(* IEC 61131-3 sources: 89152_FlorisHendrix_AfstudeerProject/89152_FlorisHendrix_ExamenProject/Stations/MachineControl/MachineControl/Class/KTS_Read, 1 file *)

(* ---- KTS_Read.st ---- *)
(*!
<Class
	Name               = "KTS_Read"
	Revision           = "0.0"
	RealtimeTask       = "true"
	DefRealtime        = "10 ms"
	CyclicTask         = "true"
	DefCyclictime      = "50 ms"
	BackgroundTask     = "false"
	Sigmatek           = "false"
	OSInterface        = "false"
	HighPriority       = "false"
	Automatic          = "false"
	UpdateMode         = "Prescan"
	SharedCommandTable = "true"
	Objectsize         = "(624,120)">
	<Channels>
		<Server Name="ClassSvr" Visualized="false" Initialize="false" WriteProtected="true" Retentive="false"/>
		<Server Name="sReadJob" Visualized="true" Initialize="false" WriteProtected="false" Retentive="false"/>
		<Server Name="sRetcode" Visualized="false" Initialize="false" WriteProtected="true" Retentive="false"/>
		<Server Name="sTeach2Points" Visualized="true" Initialize="false" WriteProtected="false" Retentive="false"/>
		<Server Name="sTeachCommand" Visualized="true" Initialize="false" WriteProtected="false" Retentive="false"/>
		<Server Name="sTeachDynamic" Visualized="true" Initialize="false" WriteProtected="false" Retentive="false"/>
		<Server Name="sTeachStart" Visualized="true" Initialize="false" WriteProtected="false" Retentive="false"/>
		<Client Name="coCSVFile" Required="true" Internal="false"/>
		<Client Name="SDCI_Device" Required="true" Internal="false"/>
		<Client Name="SDCI_Device_Async" Required="true" Internal="false"/>
		<Client Name="StringProductName" Required="true" Internal="true"/>
		<Client Name="StringVendorName" Required="true" Internal="true"/>
	</Channels>
	<Network Name="KTS_Read">
		<!-- List of Components in this network -->
		<Components>
			<Object
				Name       = "StringProductName"
				Class      = "StringRAM"
				Position   = "(180,840)"
				Visualized = "true"
				Remotely   = "true">
				<Channels>
					<Server Name="Data"/>
					<Client Name="SingleRealloc" Value="1"/>
					<Client Name="UseFile"/>
				</Channels>
			</Object>
			<Object
				Name       = "StringVendorName"
				Class      = "StringRAM"
				Position   = "(180,630)"
				Visualized = "true"
				Remotely   = "true">
				<Channels>
					<Server Name="Data"/>
					<Client Name="SingleRealloc" Value="1"/>
					<Client Name="UseFile"/>
				</Channels>
			</Object>
		</Components>
		<Comments>
		</Comments>
		<!-- List of Connections in this network -->
		<Connections>
			<Connection Source="this.StringVendorName" Destination="StringVendorName.Data"/>
			<Connection Source="this.StringProductName" Destination="StringProductName.Data"/>
		</Connections>
		<!-- Headerfiles -->
		<Options>
		</Options>
	</Network>
</Class>
*)
KTS_Read : CLASS
	TYPE
#pragma pack(push, 1)
	  UDT_KTS_Colors : STRUCT
	    Color_Red : UINT;
	    Color_Green : UINT;
	    Color_Blue : UINT;
	  END_STRUCT;
#pragma pack(pop)
#pragma pack(push, 1)
	  UDT_KTS_Color_Switch : STRUCT
	    Switch_Red : BYTE;
	    Switch_Green : BYTE;
	    Switch_Blue : BYTE;
	  END_STRUCT;
#pragma pack(pop)
#pragma pack(push, 1)
	  UDT_JobData : STRUCT
	    jd_00_Version : UINT;
	    jd_TeachLight : UDT_KTS_Colors;
	    jd_TeachDark : UDT_KTS_Colors;
	    jd_Switching_threshold : UDT_KTS_Colors;
	    jd_LD_Switches : UDT_KTS_Color_Switch;
	    jd_23_Emission_Color_KT : BYTE;
	    jd_24_Intensification_Setting_TeachIn : BYTE;
	    jd_25_Threshold_Adjustment : BYTE;
	    jd_26_Teach_Mode : BYTE;
	    jd_27_Reserved : BYTE;
	    jd_28_EmisionColor : BYTE;
	    jd_29_Switchpoint_logic : BYTE;
	    jd_30_Switchpoint_mode : BYTE;
	    jd_31_Sensitivity : BYTE;
	    jd_32_Threshold_adjustment : BYTE;
	    jd_33_Process_quality_alarm_threshold : BYTE;
	  END_STRUCT;
#pragma pack(pop)
	  UDT_KTS_TeachCommand :  //! <Type Public="true" Name="UDT_KTS_TeachCommand"/>
	  (
	    teach_1_Point_CS:=65,
	    teach_2_Points_KT_1:=67,
	    teach_2_points_KT_2:=68,
	    teach_Dynamic_KT_Start:=71,
	    teach_Dynamic_KT_Stop:=72,
	    teach_JobRead:=209
	  )$UDINT;
	  UDT_ReadJob :
	  (
	    ReadJob_Idle,
	    ReadJob_Init,
	    ReadJob_Start,
	    ReadJob_Wait,
	    ReadJob_Finish
	  )$UDINT;
	END_TYPE
  //Servers:
	ClassSvr 	: SvrChCmd_DINT;
	sRetcode 	: SvrCh_t_SDCIRetCode_PTofCls_SdiasSDCIMaster;
	sTeachStart 	: SvrCh_DINT;
	sTeachCommand 	: SvrCh_UDT_KTS_TeachCommand_PTofCls_KTS_Read;
	sTeachDynamic 	: SvrCh_DINT;
	sTeach2Points 	: SvrCh_DINT;
	sReadJob 	: SvrCh_DINT;
  //Clients:
	SDCI_Device 	: CltChCmd_SDCIDevice;
	SDCI_Device_Async 	: CltChCmd_SDCIDevice_AsyncPara;
	StringVendorName 	: CltChCmd_StringRAM;
	StringProductName 	: CltChCmd_StringRAM;
	coCSVFile 	: CltChCmd_FileBaseCsv;
  //Variables:
		vParamUINT8 	: UINT;
		vJobReadState 	: UDT_ReadJob;
		vJobData 	: UDT_JobData;
		vCsvHandle 	: DINT;
		TxtLine : ARRAY [0..255] OF CHAR;

  //Functions:

	FUNCTION VIRTUAL GLOBAL Init;

	FUNCTION VIRTUAL GLOBAL CyWork
		VAR_INPUT
			EAX 	: UDINT;
		END_VAR
		VAR_OUTPUT
			state (EAX) 	: UDINT;
		END_VAR;

	FUNCTION VIRTUAL GLOBAL RtWork
		VAR_INPUT
			EAX 	: UDINT;
		END_VAR
		VAR_OUTPUT
			state (EAX) 	: UDINT;
		END_VAR;

	FUNCTION ReadJob;

	FUNCTION CallBackReadJob
		VAR_INPUT
			pThis 	: pVoid;
			AsyState 	: SdiasSDCIMaster::t_SDCIRetCode;
			LengthOfData 	: USINT;
			pData 	: ^USINT;
		END_VAR;

	FUNCTION Swap2Bytes
		VAR_INPUT
			uiValue 	: UINT;
		END_VAR
		VAR_OUTPUT
			uiRetVal 	: UINT;
		END_VAR;

	FUNCTION SwapColors
		VAR_INPUT
			ColorsIn 	: UDT_KTS_Colors;
		END_VAR
		VAR_OUTPUT
			ColorsOut 	: UDT_KTS_Colors;
		END_VAR;

	FUNCTION WriteCsvFile;

	FUNCTION WriteCsvLine
		VAR_INPUT
			JobValue 	: DINT;
		END_VAR;

	FUNCTION VIRTUAL GLOBAL sTeachStart::Write
		VAR_INPUT
			input (EAX) 	: DINT;
		END_VAR
		VAR_OUTPUT
			result (EAX) 	: DINT;
		END_VAR;

	FUNCTION VIRTUAL GLOBAL sTeachDynamic::Write
		VAR_INPUT
			input (EAX) 	: DINT;
		END_VAR
		VAR_OUTPUT
			result (EAX) 	: DINT;
		END_VAR;

	FUNCTION VIRTUAL GLOBAL sTeach2Points::Write
		VAR_INPUT
			input (EAX) 	: DINT;
		END_VAR
		VAR_OUTPUT
			result (EAX) 	: DINT;
		END_VAR;

	FUNCTION VIRTUAL GLOBAL sReadJob::Write
		VAR_INPUT
			input (EAX) 	: DINT;
		END_VAR
		VAR_OUTPUT
			result (EAX) 	: DINT;
		END_VAR;
  //Tables:
	FUNCTION @STD
		VAR_OUTPUT
			ret_code	: CONFSTATES;
		END_VAR;
	FUNCTION GLOBAL TAB @CT_;
END_CLASS;

#pragma using StringRAM
#pragma usingLtd FileBaseCsv
#pragma usingLtd SDCIDevice
#pragma usingLtd SDCIDevice_AsyncPara

FUNCTION VIRTUAL GLOBAL KTS_Read::CyWork
	VAR_INPUT
		EAX 	: UDINT;
	END_VAR
	VAR_OUTPUT
		state (EAX) 	: UDINT;
	END_VAR

  ReadJob();

  state := READY;

END_FUNCTION

FUNCTION VIRTUAL GLOBAL KTS_Read::RtWork
	VAR_INPUT
		EAX 	: UDINT;
	END_VAR
	VAR_OUTPUT
		state (EAX) 	: UDINT;
	END_VAR

  state := READY;

END_FUNCTION

FUNCTION VIRTUAL GLOBAL KTS_Read::Init
if _FirstScan then
  vParamUINT8 := 0;
  sRetcode := SDCI_Device.SetAsyPara(ParaIndex:=0x44, ParaSubIndex:=0, WriteDataLength:=1, pWriteData:=#vParamUINT8);
end_if;
END_FUNCTION

FUNCTION VIRTUAL GLOBAL KTS_Read::sTeachStart::Write
	VAR_INPUT
		input (EAX) 	: DINT;
	END_VAR
	VAR_OUTPUT
		result (EAX) 	: DINT;
	END_VAR

	sTeachStart := input;
  if sTeachStart = 1 then
    SDCI_Device.SetAsyPara(ParaIndex:=2, ParaSubIndex:=0, WriteDataLength:=1, pWriteData:=#sTeachCommand);
  end_if;
	result := sTeachStart;

END_FUNCTION

FUNCTION VIRTUAL GLOBAL KTS_Read::sTeachDynamic::Write
	VAR_INPUT
		input (EAX) 	: DINT;
	END_VAR
	VAR_OUTPUT
		result (EAX) 	: DINT;
	END_VAR

	sTeachDynamic := input;
  if sTeachDynamic = 1 then
    sTeachCommand := teach_Dynamic_KT_Start;
  else
    sTeachCommand := teach_Dynamic_KT_Stop;
  end_if;
  sTeachStart.Write(1);

	result := sTeachDynamic;

END_FUNCTION

FUNCTION VIRTUAL GLOBAL KTS_Read::sTeach2Points::Write
	VAR_INPUT
		input (EAX) 	: DINT;
	END_VAR
	VAR_OUTPUT
		result (EAX) 	: DINT;
	END_VAR

	sTeach2Points := input;
  if sTeach2Points = 1 then
    sTeachCommand := teach_2_Points_KT_1;
  else
    sTeachCommand := teach_2_Points_KT_2;
  end_if;
  sTeachStart.Write(1);

	result := sTeach2Points;

END_FUNCTION

FUNCTION KTS_Read::ReadJob
  case vJobReadState of
    ReadJob_Init:
      sTeachCommand := teach_JobRead;
      sRetcode := SDCI_Device.SetAsyPara(ParaIndex:=2, ParaSubIndex:=0, WriteDataLength:=1, pWriteData:=#sTeachCommand);
      if sRetcode = SDCI_Ready_Ok then
        vJobReadState := ReadJob_Start;
      end_if;

    ReadJob_Start:
      sRetcode := SDCI_Device.GetAsyParaBuffered(
          ParaIndex         := 222,
          ParaSubIndex      := 0,
          pThis             := this,
          pCallBackFunction := #CallBackReadJob());
      if sRetcode = SDCI_Ready_Ok then
        vJobReadState := ReadJob_Wait;
      end_if;

    ReadJob_Wait:

    ReadJob_Finish:
      vJobReadState := ReadJob_Idle;

  end_case;
END_FUNCTION

FUNCTION KTS_Read::CallBackReadJob
	VAR_INPUT
		pThis 	: pVoid;
		AsyState 	: SdiasSDCIMaster::t_SDCIRetCode;
		LengthOfData 	: USINT;
		pData 	: ^USINT;
	END_VAR

  THIS := pThis$^KTS_Read;

  if AsyState = SdiasSDCIMaster::t_SDCIRetCode::SDCI_Ready_Ok then

    if LengthOfData > 0 & pData then

      if LengthOfData <= sizeof(UDT_JobData) then
        _memcpy(ptr1:=#vJobData, ptr2:=pData, cntr:=LengthOfData);

        vJobData.jd_TeachLight := SwapColors(vJobData.jd_TeachLight);
        vJobData.jd_TeachDark := SwapColors(vJobData.jd_TeachDark);
        vJobData.jd_Switching_threshold := SwapColors(vJobData.jd_Switching_threshold);
      end_if;

    end_if;

    WriteCsvFile();
  end_if;
  vJobReadState := ReadJob_Finish;

END_FUNCTION

FUNCTION VIRTUAL GLOBAL KTS_Read::sReadJob::Write
	VAR_INPUT
		input (EAX) 	: DINT;
	END_VAR
	VAR_OUTPUT
		result (EAX) 	: DINT;
	END_VAR

	sReadJob := input;
  if sReadJob = 1 then
    vJobReadState := ReadJob_Init;
  end_if;
	result := sReadJob;

END_FUNCTION

FUNCTION KTS_Read::Swap2Bytes
	VAR_INPUT
		uiValue 	: UINT;
	END_VAR
	VAR_OUTPUT
		uiRetVal 	: UINT;
	END_VAR

  uiRetVal := 0x0000;
  uiRetVal := uiRetVal OR ((uiValue AND 0x00FF) SHL 8);
  uiRetVal := uiRetVal OR ((uiValue AND 0xFF00) SHR 8);

END_FUNCTION

FUNCTION KTS_Read::SwapColors
	VAR_INPUT
		ColorsIn 	: UDT_KTS_Colors;
	END_VAR
	VAR_OUTPUT
		ColorsOut 	: UDT_KTS_Colors;
	END_VAR
  ColorsOut.Color_Red := Swap2Bytes(ColorsIn.Color_Red);
  ColorsOut.Color_Green := Swap2Bytes(ColorsIn.Color_Green);
  ColorsOut.Color_Blue := Swap2Bytes(ColorsIn.Color_Blue);
END_FUNCTION

FUNCTION KTS_Read::WriteCsvFile

  vCsvHandle := coCSVFile.OpenFile(filename:="C:\\kts\\textcsv.csv", attrib:=ATT_CREATE_ALWAYS);
 	if vCsvHandle <= 0 then
    return;
  end_if;

  WriteCsvLine(vJobData.jd_00_Version);
  WriteCsvLine(vJobData.jd_TeachLight.Color_Red);
  WriteCsvLine(vJobData.jd_TeachLight.Color_Green);
  WriteCsvLine(vJobData.jd_TeachLight.Color_Blue);
  WriteCsvLine(vJobData.jd_TeachDark.Color_Red);
  WriteCsvLine(vJobData.jd_TeachDark.Color_Green);
  WriteCsvLine(vJobData.jd_TeachDark.Color_Blue);
  WriteCsvLine(vJobData.jd_Switching_threshold.Color_Red);
  WriteCsvLine(vJobData.jd_Switching_threshold.Color_Green);
  WriteCsvLine(vJobData.jd_Switching_threshold.Color_Blue);
  WriteCsvLine(vJobData.jd_LD_Switches.Switch_Red);
  WriteCsvLine(vJobData.jd_LD_Switches.Switch_Blue);
  WriteCsvLine(vJobData.jd_LD_Switches.Switch_Green);
  WriteCsvLine(vJobData.jd_23_Emission_Color_KT);
  WriteCsvLine(vJobData.jd_24_Intensification_Setting_TeachIn);
  WriteCsvLine(vJobData.jd_25_Threshold_Adjustment);
  WriteCsvLine(vJobData.jd_26_Teach_Mode);
  WriteCsvLine(vJobData.jd_27_Reserved);
  WriteCsvLine(vJobData.jd_28_EmisionColor);
  WriteCsvLine(vJobData.jd_29_Switchpoint_logic);
  WriteCsvLine(vJobData.jd_30_Switchpoint_mode);
  WriteCsvLine(vJobData.jd_31_Sensitivity);
  WriteCsvLine(vJobData.jd_32_Threshold_adjustment);
  WriteCsvLine(vJobData.jd_33_Process_quality_alarm_threshold);

  coCSVFile.CloseFile(handle:=vCsvHandle);

END_FUNCTION

FUNCTION KTS_Read::WriteCsvLine
	VAR_INPUT
		JobValue 	: DINT;
	END_VAR
  VAR
    offset : DINT;
  END_VAR

  offset:= coCSVFile.BuildValue2Ascii(value:= JobValue$DINT, dest:= #TxtLine[0], offset:= 0);
  offset+= coCSVFile.BuildEol(dest:= #TxtLine[0], offset:= offset);

  coCSVFile.WriteLine(handle:= vCsvHandle, src:= #TxtLine[0], len:= offset);

END_FUNCTION
